// TIA Portal V17 export
// export: Created 2025-06-25T13:13:07.163732Z, ExportSetting WithDefaults, DisplayName Totally Integrated Automation Portal, DisplayVersion V17 Update 8, DisplayName TIA Portal Openness, DisplayVersion V17 Update 8, DisplayName TIA Portal Version Control Interface, DisplayVersion V17, DisplayName STEP 7 Professional, DisplayVersion V17 Update 8, DisplayName STEP 7 Safety, DisplayVersion V17 Update 6, DisplayName WinCC Advanced, DisplayVersion V17 Update 8
FUNCTION_BLOCK "CrankcasePressureControl"   // FB2, FBD
TITLE = Crankcase pressure control system (CPC)
{ S7_Optimized_Access := 'TRUE' }
VERSION : 0.1
// stored: AutoNumber true, IsIECCheckEnabled false, IsRetainMemResEnabled false, MemoryReserve 100, SetENOAutomatically false, UDAEnableTagReadback false
   VAR_INPUT
      bEnable { ExternalAccessible := 'False'; ExternalVisible := 'False'; ExternalWritable := 'False'} : Bool;
      bReset { ExternalAccessible := 'False'; ExternalVisible := 'False'; ExternalWritable := 'False'} : Bool;   // 1 = reset manual modes
   END_VAR
   VAR_OUTPUT
      bPumpOut { ExternalAccessible := 'False'; ExternalVisible := 'False'; ExternalWritable := 'False'} : Bool;   // 1 = run pump, 0 = do not run pump
   END_VAR
   VAR
      Cooler { ExternalAccessible := 'False'; ExternalVisible := 'False'; ExternalWritable := 'False'; S7_SetPoint := 'True'} : "fbPI_Regulator";
      LevelControl { ExternalAccessible := 'False'; ExternalVisible := 'False'; ExternalWritable := 'False'; S7_SetPoint := 'True'} : "fbOnOffRegulator";   // Regulate level based on direct level measurement
      LevelControl2 { ExternalAccessible := 'False'; ExternalVisible := 'False'; ExternalWritable := 'False'; S7_SetPoint := 'True'} : "fbProgressivePeriodicRegulator4";
      HighAlarm { ExternalAccessible := 'False'; ExternalVisible := 'False'; ExternalWritable := 'False'; S7_SetPoint := 'True'} : "fbHighAlarm";
   END_VAR
   VAR_TEMP
      bPumpOut1 : Bool;
      bPumpOut2 : Bool;
   END_VAR
BEGIN

REGION Network 1: Cooling fan regulator
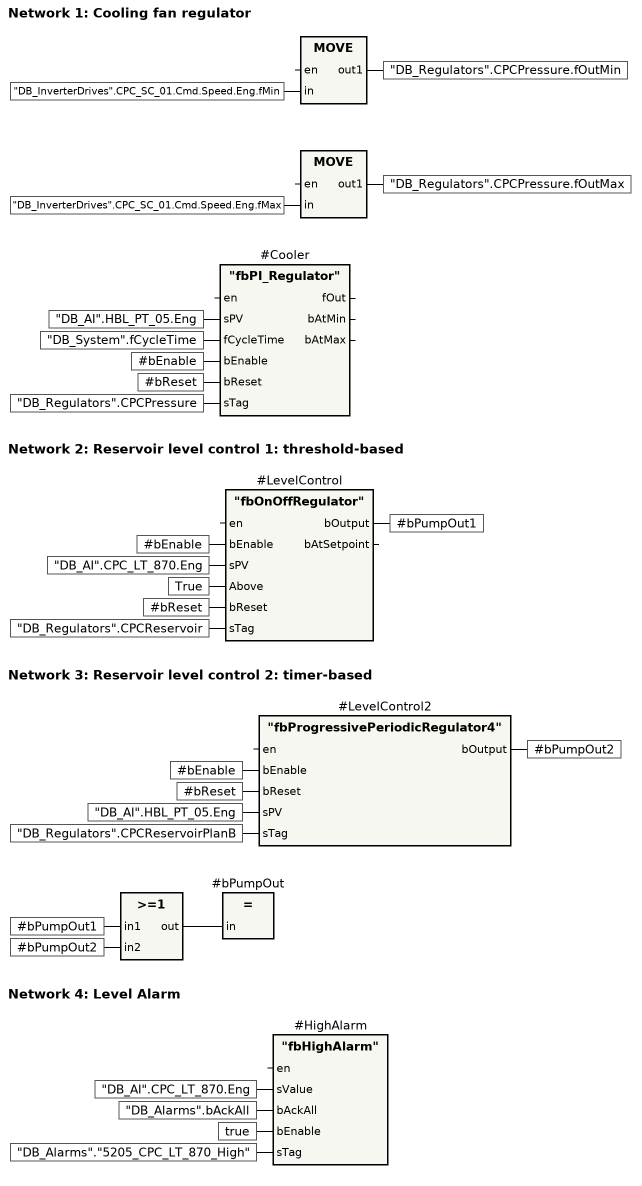
   "DB_Regulators".CPCPressure.fOutMin := "DB_InverterDrives".CPC_SC_01.Cmd.Speed.Eng.fMin;
   "DB_Regulators".CPCPressure.fOutMax := "DB_InverterDrives".CPC_SC_01.Cmd.Speed.Eng.fMax;
   #Cooler(sPV := "DB_AI".HBL_PT_05.Eng,   // "fbPI_Regulator"
           fCycleTime := "DB_System".fCycleTime,
           bEnable := #bEnable,
           bReset := #bReset,
           sTag := "DB_Regulators".CPCPressure);
END_REGION

REGION Network 2: Reservoir level control 1: threshold-based
   #LevelControl(bEnable := #bEnable,   // "fbOnOffRegulator"
                 sPV := "DB_AI".CPC_LT_870.Eng,
                 Above := True,
                 bReset := #bReset,
                 sTag := "DB_Regulators".CPCReservoir,
                 bOutput => #bPumpOut1);
END_REGION

REGION Network 3: Reservoir level control 2: timer-based
   #LevelControl2(bEnable := #bEnable,   // "fbProgressivePeriodicRegulator4"
                  bReset := #bReset,
                  sPV := "DB_AI".HBL_PT_05.Eng,
                  sTag := "DB_Regulators".CPCReservoirPlanB,
                  bOutput => #bPumpOut2);
   #bPumpOut := #bPumpOut1 OR #bPumpOut2;
END_REGION

REGION Network 4: Level Alarm
   #HighAlarm(sValue := "DB_AI".CPC_LT_870.Eng,   // "fbHighAlarm"
              bAckAll := "DB_Alarms".bAckAll,
              bEnable := true,
              sTag := "DB_Alarms"."5205_CPC_LT_870_High");
END_REGION
END_FUNCTION_BLOCK
